//----------------------------------------------------------------------------//
//            Copyright 2018 Rieckermann Engineering Operations               //
//----------------------------------------------------------------------------//
// Class:       fcDI3                                                         //
// Description:                                                               //
// General alarm single digital input.                                        //
//----------------------------------------------------------------------------//
// Revision history:                                                          //
// Rev By               Date        CC        Note                            //
// 1.0 David Paspa      17-Apr-2018 NA        Initial design from DI1.        //
//----------------------------------------------------------------------------//
FUNCTION "fcDI3" : Void
TITLE = DI3 : General alarm with software input
{ S7_Optimized_Access := 'TRUE' }
NAME : fcDI3
AUTHOR : REO
VERSION : 1.0

//----------------------------------------------------------------------------//
// Declare variables:                                                         //
//----------------------------------------------------------------------------//
VAR_IN_OUT
    p : "udtDI3";            // Block data interface
END_VAR

VAR_TEMP
    tPV : Bool;              // Temporary processed DI signal
END_VAR

BEGIN
NETWORK
TITLE = Call Mode and Command handling function
    //------------------------------------------------------------------------//
    // MODE AND COMMAND   MODE AND COMMAND   MODE AND COMMAND   MODE AND COMM //
    // MODE AND COMMAND   MODE AND COMMAND   MODE AND COMMAND   MODE AND COMM //
    //                                                                        //
    // Process the standard block functions for command, mode, interlock and  //
    // state:                                                                 //
    //------------------------------------------------------------------------//
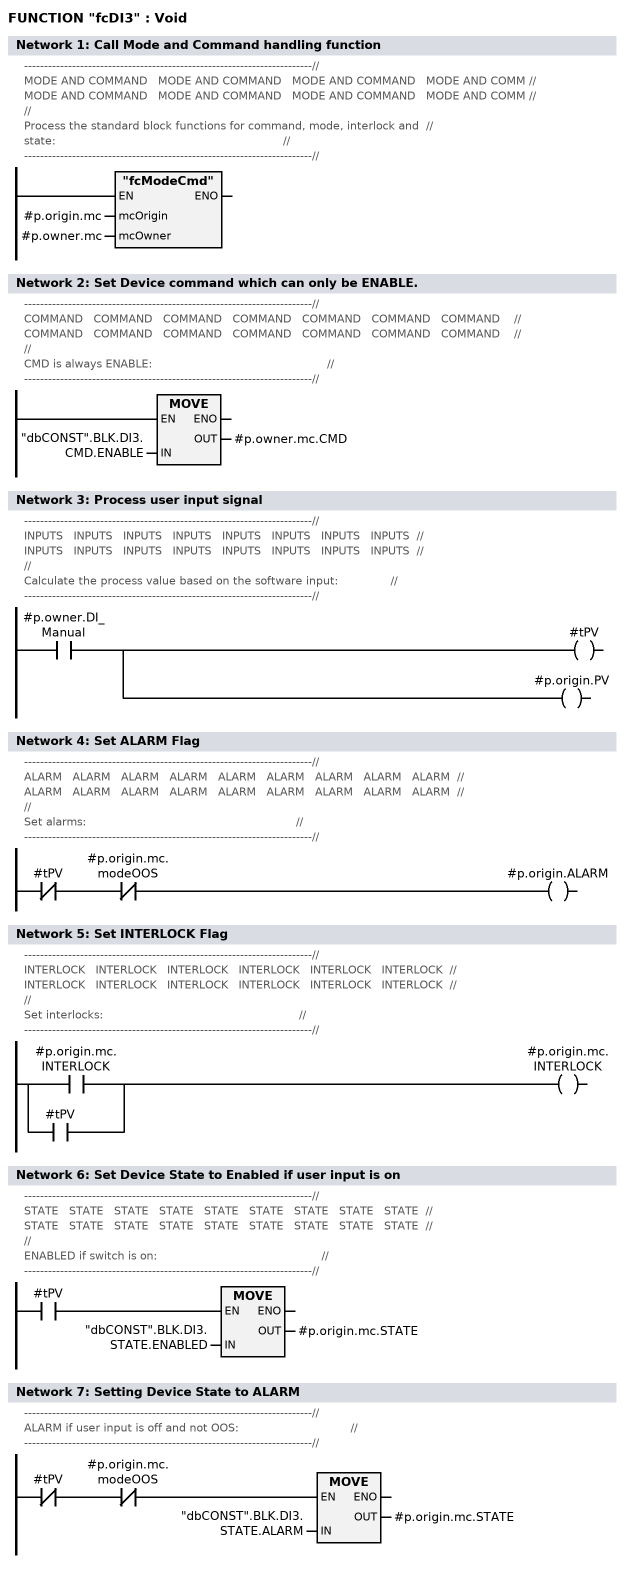
    CALL "fcModeCmd"
    (   mcOrigin             := #p.origin.mc ,
        mcOwner              := #p.owner.mc
    );

NETWORK
TITLE = Set Device command which can only be ENABLE.
    //------------------------------------------------------------------------//
    // COMMAND   COMMAND   COMMAND   COMMAND   COMMAND   COMMAND   COMMAND    //
    // COMMAND   COMMAND   COMMAND   COMMAND   COMMAND   COMMAND   COMMAND    //
    //                                                                        //
    // CMD is always ENABLE:                                                  //
    //------------------------------------------------------------------------//
    L "dbCONST".BLK.DI3.CMD.ENABLE;
    T #p.owner.mc.CMD;

NETWORK
TITLE = Process user input signal
    //------------------------------------------------------------------------//
    // INPUTS   INPUTS   INPUTS   INPUTS   INPUTS   INPUTS   INPUTS   INPUTS  //
    // INPUTS   INPUTS   INPUTS   INPUTS   INPUTS   INPUTS   INPUTS   INPUTS  //
    //                                                                        //
    // Calculate the process value based on the software input:               //
    //------------------------------------------------------------------------//
    A #p.owner.DI_Manual;
    = #tPV;
    = #p.origin.PV;

NETWORK
TITLE = Set ALARM Flag
    //------------------------------------------------------------------------//
    // ALARM   ALARM   ALARM   ALARM   ALARM   ALARM   ALARM   ALARM   ALARM  //
    // ALARM   ALARM   ALARM   ALARM   ALARM   ALARM   ALARM   ALARM   ALARM  //
    //                                                                        //
    // Set alarms:                                                            //
    //------------------------------------------------------------------------//
    AN #tPV;
    AN #p.origin.mc.modeOOS;
    = #p.origin.ALARM;

NETWORK
TITLE = Set INTERLOCK Flag
    //------------------------------------------------------------------------//
    // INTERLOCK   INTERLOCK   INTERLOCK   INTERLOCK   INTERLOCK   INTERLOCK  //
    // INTERLOCK   INTERLOCK   INTERLOCK   INTERLOCK   INTERLOCK   INTERLOCK  //
    //                                                                        //
    // Set interlocks:                                                        //
    //------------------------------------------------------------------------//
    O #p.origin.mc.INTERLOCK;
    O #tPV;
    = #p.origin.mc.INTERLOCK;

NETWORK
TITLE = Set Device State to Enabled if user input is on
    //------------------------------------------------------------------------//
    // STATE   STATE   STATE   STATE   STATE   STATE   STATE   STATE   STATE  //
    // STATE   STATE   STATE   STATE   STATE   STATE   STATE   STATE   STATE  //
    //                                                                        //
    // ENABLED if switch is on:                                               //
    //------------------------------------------------------------------------//
    A #tPV;
    JCN _a;
    L "dbCONST".BLK.DI3.STATE.ENABLED;
    T #p.origin.mc.STATE;
_a:   NOP 0;

NETWORK
TITLE = Setting Device State to ALARM
    //------------------------------------------------------------------------//
    // ALARM if user input is off and not OOS:                                //
    //------------------------------------------------------------------------//
    AN #tPV;
    AN #p.origin.mc.modeOOS;
    JCN _b;
    L "dbCONST".BLK.DI3.STATE.ALARM;
    T #p.origin.mc.STATE;
_b:   NOP 0;
END_FUNCTION
